// ============================================
// DB_RecipeProgram3 - Program 3
// Lines: 97
// CHUNKS: 5 x 100
// Generated by SpinningCam  [2026-09-29 00:05:30]
// !!! CONTINUOUS MOTION (CMD=2) - EXPERIMENTAL PLC ONLY !!!
// Load ONLY on the continuous-motion PLC build. A production PLC
// skips CMD=2 lines and jumps straight between the other points.
// T=0.045 s, corner tol=0.2 mm, F min=180, exact stop at >= 90 deg, stop slow-down=OFF
// CMD=2 lines: 76, exact corners: 0, slowed corners: 7 (+11 leaving), slowed stops: 0
// ============================================
//
// --- MAKINE AYARLARI ---
// Machine Origin  : X=0.0, Z=0.0
// Axis Direction  : X=NORMAL, Z=NORMAL
// Output Mode     : RADIUS
// G54 Offset      : X=0.0, Z=0.0
// Home            : X=-394.0, Z=-174.0
// Retract         : X=-10.0, Z=-10.0
//
// --- PARCA / BLANK ---
// Blank Radius    : 77.8 mm
// Blank Z Shift   : 0.0 mm
// Final Thickness : 0.8 mm
// Min Safety Gap  : 0.0 mm
//
// --- MANDREL POZISYON ---
// Mandrel Offset  : X=0.0, Z=0.0
// Mandrel Rot     : Rx=90.0, Ry=0.0, Rz=0.0
//
// --- OPERASYONLAR ---
// Op1: ROUGHING, 1 paso, T004, R=44.56mm, RPM=600.0, mm_min=900.0
// Op2: ROUGHING, 1 paso, T004, R=44.56mm, RPM=600.0, mm_min=900.0
// Op3: ROUGHING, 1 paso, T004, R=44.56mm, RPM=600.0, mm_min=900.0
// Op4: ROUGHING, 1 paso, T004, R=44.56mm, RPM=600.0, mm_min=900.0
// Op5: ROUGHING, 1 paso, T004, R=44.56mm, RPM=600.0, mm_min=900.0
// Op6: ROUGHING, 1 paso, T004, R=44.56mm, RPM=600.0, mm_min=800.0
// Op7: ROUGHING, 1 paso, T004, R=44.56mm, RPM=600.0, mm_min=800.0
// Op8: ROUGHING, 1 paso, T004, R=44.56mm, RPM=600.0, mm_min=800.0
// Op9: ROUGHING, 1 paso, T004, R=44.56mm, RPM=600.0, mm_min=800.0
// Op10: ROUGHING, 1 paso, T004, R=44.56mm, RPM=600.0, mm_min=800.0
// Op11: ROUGHING, 1 paso, T004, R=44.56mm, RPM=600.0, mm_min=800.0
// Op12: ROUGHING, 1 paso, T004, R=44.56mm, RPM=600.0, mm_min=800.0
// Op13: ROUGHING, 1 paso, T004, R=44.56mm, RPM=600.0, mm_min=1000.0
// Op14: ROUGHING, 1 paso, T004, R=44.56mm, RPM=600.0, mm_min=1000.0
// Op15: ROUGHING, 1 paso, T004, R=44.56mm, RPM=600.0, mm_min=1000.0
// Op16: ROUGHING, 1 paso, T004, R=44.56mm, RPM=600.0, mm_min=1000.0
// Op17: ROUGHING, 1 paso, T004, R=44.56mm, RPM=600.0, mm_min=1000.0
// Op18: ROUGHING, 1 paso, T004, R=44.56mm, RPM=600.0, mm_min=1000.0
// Op19: ROUGHING, 1 paso, T004, R=44.56mm, RPM=600.0, mm_min=1000.0
// Op20: ROUGHING, 1 paso, T004, R=44.56mm, RPM=600.0, mm_min=1000.0
// Op21: ROUGHING, 1 paso, T004, R=44.56mm, RPM=600.0, mm_min=1000.0
// Op22: ROUGHING, 1 paso, T004, R=44.56mm, RPM=600.0, mm_min=1000.0
// Op23: ROUGHING, 1 paso, T004, R=44.56mm, RPM=600.0, mm_min=1000.0
// Op24: ROUGHING, 1 paso, T004, R=44.56mm, RPM=600.0, mm_min=1000.0
// Op25: ROUGHING, 1 paso, T004, R=44.56mm, RPM=600.0, mm_min=1000.0
// Op26: ROUGHING, 1 paso, T004, R=44.56mm, RPM=600.0, mm_min=1000.0
// Op27: CUTTING, 1 paso, T006, R=20.0mm, RPM=500.0, mm_min=10.0
// Op28: ROUGHING, 1 paso, T004, R=44.56mm, RPM=600.0, mm_min=1000.0
// Op29: ROUGHING, 1 paso, T004, R=44.56mm, RPM=600.0, mm_min=1000.0
// Op30: ROUGHING, 1 paso, T004, R=44.56mm, RPM=600.0, mm_min=1000.0
// Op31: ROUGHING, 1 paso, T004, R=44.56mm, RPM=600.0, mm_min=1000.0
// Op32: ROUGHING, 1 paso, T004, R=44.56mm, RPM=600.0, mm_min=1000.0
// Op33: ROUGHING, 1 paso, T004, R=44.56mm, RPM=600.0, mm_min=1000.0
// Op34: ROUGHING, 1 paso, T004, R=44.56mm, RPM=600.0, mm_min=1000.0
// Op35: ROUGHING, 1 paso, T004, R=44.56mm, RPM=600.0, mm_min=1000.0
// Op36: ROUGHING, 1 paso, T004, R=44.56mm, RPM=600.0, mm_min=1500.0
// Op37: ROUGHING, 1 paso, T004, R=44.56mm, RPM=600.0, mm_min=1500.0
// Op38: ROUGHING, 1 paso, T004, R=44.56mm, RPM=600.0, mm_min=1500.0
// Op39: ROUGHING, 1 paso, T004, R=44.56mm, RPM=600.0, mm_min=1500.0
// Op40: ROUGHING, 1 paso, T004, R=44.56mm, RPM=600.0, mm_min=1500.0
// Op41: ROUGHING, 1 paso, T004, R=44.56mm, RPM=600.0, mm_min=1500.0
// Op42: ROUGHING, 1 paso, T004, R=44.56mm, RPM=600.0, mm_min=1500.0
// Op43: ROUGHING, 1 paso, T004, R=44.56mm, RPM=600.0, mm_min=1500.0
// Op44: ROUGHING, 1 paso, T004, R=44.56mm, RPM=600.0, mm_min=1500.0
// Op45: ROUGHING, 1 paso, T004, R=44.56mm, RPM=600.0, mm_min=1500.0
// Op46: ROUGHING, 1 paso, T004, R=44.56mm, RPM=600.0, mm_min=1500.0
// Op47: ROUGHING, 1 paso, T004, R=44.56mm, RPM=600.0, mm_min=1500.0
// Op48: ROUGHING, 1 paso, T004, R=44.56mm, RPM=600.0, mm_min=1500.0
// Op49: ROUGHING, 1 paso, T004, R=44.56mm, RPM=600.0, mm_min=1500.0
// Op50: ROUGHING, 1 paso, T004, R=44.56mm, RPM=600.0, mm_min=1500.0
// Op51: ROUGHING, 1 paso, T004, R=44.56mm, RPM=600.0, mm_min=1500.0
// Op52: ROUGHING, 1 paso, T004, R=44.56mm, RPM=600.0, mm_min=1500.0
// Op53: ROUGHING, 1 paso, T004, R=44.56mm, RPM=600.0, mm_min=1500.0
// Op54: ROUGHING, 1 paso, T004, R=44.56mm, RPM=600.0, mm_min=1500.0
// Op55: ROUGHING, 1 paso, T004, R=44.56mm, RPM=600.0, mm_min=1500.0
// Op56: ROUGHING, 1 paso, T004, R=44.56mm, RPM=600.0, mm_min=1500.0
// Op57: ROUGHING, 1 paso, T004, R=44.56mm, RPM=600.0, mm_min=1500.0
// Op58: ROUGHING, 1 paso, T004, R=44.56mm, RPM=600.0, mm_min=1500.0
// Op59: ROUGHING, 1 paso, T004, R=44.56mm, RPM=600.0, mm_min=1500.0
// Op60: ROUGHING, 1 paso, T004, R=44.56mm, RPM=800.0, mm_min=1500.0
// Op61: ROUGHING, 1 paso, T004, R=44.56mm, RPM=800.0, mm_min=800.0
// Op62: ROUGHING, 1 paso, T004, R=44.56mm, RPM=800.0, mm_min=800.0
// Op63: ROUGHING, 1 paso, T004, R=44.56mm, RPM=600.0, mm_min=1500.0
// Op64: ROUGHING, 1 paso, T004, R=44.56mm, RPM=600.0, mm_min=1500.0
// Op65: ROUGHING, 1 paso, T004, R=44.56mm, RPM=600.0, mm_min=1500.0
// Op66: ROUGHING, 1 paso, T004, R=44.56mm, RPM=600.0, mm_min=1500.0
// Op67: ROUGHING, 1 paso, T004, R=44.56mm, RPM=600.0, mm_min=1500.0
// Op68: ROUGHING, 1 paso, T004, R=44.56mm, RPM=600.0, mm_min=1500.0
// Op69: ROUGHING, 1 paso, T004, R=44.56mm, RPM=600.0, mm_min=1500.0
// Op70: ROUGHING, 1 paso, T004, R=44.56mm, RPM=600.0, mm_min=1500.0
// Op71: ROUGHING, 1 paso, T004, R=44.56mm, RPM=600.0, mm_min=1500.0
// Op72: ROUGHING, 1 paso, T004, R=44.56mm, RPM=600.0, mm_min=1000.0
// Op73: ROUGHING, 1 paso, T004, R=44.56mm, RPM=600.0, mm_min=1000.0
// Op74: ROUGHING, 1 paso, T004, R=44.56mm, RPM=600.0, mm_min=1000.0
// Op75: ROUGHING, 1 paso, T004, R=44.56mm, RPM=600.0, mm_min=1000.0
// Op76: ROUGHING, 1 paso, T004, R=44.56mm, RPM=600.0, mm_min=1500.0
// Op77: ROUGHING, 1 paso, T004, R=44.56mm, RPM=600.0, mm_min=1000.0
// Op78: ROUGHING, 1 paso, T004, R=44.56mm, RPM=600.0, mm_min=1000.0
// Op79: ROUGHING, 1 paso, T004, R=44.56mm, RPM=600.0, mm_min=1000.0
// Op80: ROUGHING, 1 paso, T004, R=44.56mm, RPM=600.0, mm_min=1000.0
// Op81: ROUGHING, 1 paso, T004, R=44.56mm, RPM=600.0, mm_min=1000.0
// Op82: ROUGHING, 1 paso, T004, R=44.56mm, RPM=600.0, mm_min=1000.0
// Op83: ROUGHING, 1 paso, T004, R=44.56mm, RPM=600.0, mm_min=1000.0
// Op84: ROUGHING, 1 paso, T004, R=44.56mm, RPM=600.0, mm_min=1000.0
// Op85: ROUGHING, 1 paso, T004, R=44.56mm, RPM=600.0, mm_min=1000.0
// Op86: ROUGHING, 1 paso, T004, R=44.56mm, RPM=600.0, mm_min=1000.0
// Op87: ROUGHING, 1 paso, T004, R=44.56mm, RPM=600.0, mm_min=1000.0
// Op88: ROUGHING, 1 paso, T004, R=44.56mm, RPM=600.0, mm_min=1000.0
// Op89: ROUGHING, 1 paso, T004, R=44.56mm, RPM=600.0, mm_min=1000.0
// Op90: ROUGHING, 1 paso, T004, R=44.56mm, RPM=600.0, mm_min=1000.0
// Op91: ROUGHING, 1 paso, T004, R=44.56mm, RPM=600.0, mm_min=1000.0
// Op92: ROUGHING, 1 paso, T004, R=44.56mm, RPM=600.0, mm_min=1000.0
// Op93: ROUGHING, 1 paso, T004, R=44.56mm, RPM=600.0, mm_min=1000.0
// Op94: ROUGHING, 1 paso, T004, R=44.56mm, RPM=600.0, mm_min=1000.0
// Op95: ROUGHING, 1 paso, T004, R=44.56mm, RPM=600.0, mm_min=1000.0
// Op96: ROUGHING, 1 paso, T004, R=44.56mm, RPM=600.0, mm_min=1000.0
// Op97: ROUGHING, 1 paso, T004, R=44.56mm, RPM=600.0, mm_min=1000.0
// Op98: ROUGHING, 1 paso, T004, R=44.56mm, RPM=600.0, mm_min=1000.0
// Op99: ROUGHING, 1 paso, T004, R=44.56mm, RPM=600.0, mm_min=1000.0
// Op100: ROUGHING, 1 paso, T004, R=44.56mm, RPM=600.0, mm_min=1000.0
// Op101: ROUGHING, 1 paso, T004, R=44.56mm, RPM=600.0, mm_min=1000.0
// Op102: ROUGHING, 1 paso, T004, R=44.56mm, RPM=600.0, mm_min=1000.0
// Op103: ROUGHING, 1 paso, T004, R=44.56mm, RPM=600.0, mm_min=1000.0
// Op104: ROUGHING, 1 paso, T004, R=44.56mm, RPM=600.0, mm_min=1000.0
// Op105: ROUGHING, 1 paso, T004, R=44.56mm, RPM=600.0, mm_min=1000.0
// Op106: ROUGHING, 1 paso, T004, R=44.56mm, RPM=600.0, mm_min=1000.0
// Op107: ROUGHING, 1 paso, T004, R=44.56mm, RPM=600.0, mm_min=1000.0
// Op108: ROUGHING, 1 paso, T004, R=44.56mm, RPM=600.0, mm_min=1000.0
// Op109: ROUGHING, 1 paso, T004, R=44.56mm, RPM=600.0, mm_min=1000.0
// Op110: ROUGHING, 1 paso, T004, R=44.56mm, RPM=600.0, mm_min=1000.0
// Op111: ROUGHING, 1 paso, T004, R=44.56mm, RPM=600.0, mm_min=1000.0
// Op112: ROUGHING, 1 paso, T004, R=44.56mm, RPM=600.0, mm_min=1000.0
// Op113: ROUGHING, 1 paso, T004, R=44.56mm, RPM=600.0, mm_min=1000.0
// Op114: ROUGHING, 1 paso, T004, R=44.56mm, RPM=600.0, mm_min=1000.0
// Op115: ROUGHING, 1 paso, T004, R=44.56mm, RPM=600.0, mm_min=1000.0
// Op116: ROUGHING, 1 paso, T004, R=44.56mm, RPM=600.0, mm_min=1000.0
// Op117: ROUGHING, 1 paso, T004, R=44.56mm, RPM=600.0, mm_min=1000.0
// Op118: ROUGHING, 1 paso, T004, R=44.56mm, RPM=600.0, mm_min=1000.0
// Op119: ROUGHING, 1 paso, T004, R=44.56mm, RPM=600.0, mm_min=1000.0
// Op120: ROUGHING, 1 paso, T004, R=44.56mm, RPM=600.0, mm_min=1000.0
// Op121: ROUGHING, 1 paso, T004, R=44.56mm, RPM=600.0, mm_min=1000.0
// Op122: ROUGHING, 1 paso, T004, R=44.56mm, RPM=600.0, mm_min=1000.0
// Op123: ROUGHING, 1 paso, T004, R=44.56mm, RPM=600.0, mm_min=1000.0
// Op124: ROUGHING, 1 paso, T004, R=44.56mm, RPM=600.0, mm_min=1000.0
// Op125: ROUGHING, 1 paso, T004, R=44.56mm, RPM=600.0, mm_min=1000.0
// Op126: ROUGHING, 1 paso, T004, R=44.56mm, RPM=600.0, mm_min=1000.0
// Op127: ROUGHING, 1 paso, T004, R=44.56mm, RPM=600.0, mm_min=1000.0
// Op128: ROUGHING, 1 paso, T004, R=44.56mm, RPM=600.0, mm_min=1000.0
// Op129: CUTTING, 1 paso, T006, R=20.0mm, RPM=500.0, mm_min=7.0
// Op130: ROUGHING, 1 paso, T004, R=44.56mm, RPM=600.0, mm_min=1000.0
// Op131: ROUGHING, 1 paso, T004, R=44.56mm, RPM=600.0, mm_min=1000.0
// Op132: ROUGHING, 1 paso, T004, R=44.56mm, RPM=600.0, mm_min=1000.0
// Op133: ROUGHING, 1 paso, T004, R=44.56mm, RPM=600.0, mm_min=1000.0
// Op134: ROUGHING, 1 paso, T004, R=44.56mm, RPM=600.0, mm_min=1000.0
// Op135: ROUGHING, 1 paso, T004, R=44.56mm, RPM=600.0, mm_min=1000.0
// Op136: ROUGHING, 1 paso, T004, R=44.56mm, RPM=600.0, mm_min=1000.0
// Op137: ROUGHING, 1 paso, T004, R=44.56mm, RPM=600.0, mm_min=400.0
// Op138: ROUGHING, 1 paso, T004, R=44.56mm, RPM=600.0, mm_min=400.0
// Op139: ROUGHING, 1 paso, T004, R=44.56mm, RPM=600.0, mm_min=400.0
// Op140: ROUGHING, 1 paso, T004, R=44.56mm, RPM=600.0, mm_min=1000.0
// Op141: ROUGHING, 1 paso, T004, R=44.56mm, RPM=600.0, mm_min=400.0
// Op142: ROUGHING, 1 paso, T004, R=44.56mm, RPM=600.0, mm_min=400.0
// Op143: ROUGHING, 1 paso, T004, R=44.56mm, RPM=600.0, mm_min=400.0
// Op144: ROUGHING, 1 paso, T004, R=44.56mm, RPM=600.0, mm_min=400.0
// Op145: ROUGHING, 1 paso, T004, R=44.56mm, RPM=600.0, mm_min=400.0
// Op146: ROUGHING, 1 paso, T004, R=44.56mm, RPM=600.0, mm_min=400.0
// Op147: ROUGHING, 1 paso, T004, R=44.56mm, RPM=600.0, mm_min=400.0
// Op148: ROUGHING, 1 paso, T004, R=44.56mm, RPM=600.0, mm_min=400.0
// Op149: ROUGHING, 1 paso, T004, R=44.56mm, RPM=600.0, mm_min=400.0
// Op150: ROUGHING, 1 paso, T004, R=44.56mm, RPM=600.0, mm_min=400.0
// Op151: ROUGHING, 1 paso, T004, R=44.56mm, RPM=600.0, mm_min=400.0
// Op152: ROUGHING, 1 paso, T004, R=44.56mm, RPM=600.0, mm_min=400.0
// Op153: ROUGHING, 1 paso, T004, R=44.56mm, RPM=600.0, mm_min=400.0
// Op154: ROUGHING, 1 paso, T004, R=44.56mm, RPM=600.0, mm_min=400.0
// Op155: ROUGHING, 1 paso, T004, R=44.56mm, RPM=600.0, mm_min=400.0
// Op156: ROUGHING, 1 paso, T004, R=44.56mm, RPM=600.0, mm_min=400.0
// Op157: ROUGHING, 1 paso, T004, R=44.56mm, RPM=600.0, mm_min=400.0
// Op158: ROUGHING, 1 paso, T004, R=44.56mm, RPM=600.0, mm_min=400.0
// Op159: ROUGHING, 1 paso, T004, R=44.56mm, RPM=600.0, mm_min=400.0
// Op160: ROUGHING, 1 paso, T004, R=44.56mm, RPM=600.0, mm_min=400.0
// Op161: ROUGHING, 1 paso, T004, R=44.56mm, RPM=600.0, mm_min=400.0
// Op162: ROUGHING, 1 paso, T004, R=44.56mm, RPM=600.0, mm_min=400.0
// Op163: ROUGHING, 1 paso, T004, R=44.56mm, RPM=600.0, mm_min=400.0
// Op164: ROUGHING, 1 paso, T004, R=44.56mm, RPM=600.0, mm_min=400.0
// Op165: ROUGHING, 1 paso, T004, R=44.56mm, RPM=600.0, mm_min=400.0
// Op166: ROUGHING, 1 paso, T004, R=44.56mm, RPM=600.0, mm_min=400.0
// Op167: ROUGHING, 1 paso, T004, R=44.56mm, RPM=800.0, mm_min=400.0
// Op168: ROUGHING, 1 paso, T004, R=44.56mm, RPM=800.0, mm_min=400.0
// Op169: ROUGHING, 1 paso, T004, R=44.56mm, RPM=800.0, mm_min=400.0
// Op170: ROUGHING, 1 paso, T004, R=44.56mm, RPM=800.0, mm_min=400.0
// Op171: ROUGHING, 1 paso, T004, R=44.56mm, RPM=800.0, mm_min=400.0
// Op172: ROUGHING, 1 paso, T004, R=44.56mm, RPM=800.0, mm_min=400.0
// Op173: ROUGHING, 1 paso, T004, R=44.56mm, RPM=800.0, mm_min=400.0
// Op174: ROUGHING, 1 paso, T004, R=44.56mm, RPM=800.0, mm_min=400.0
// Op175: ROUGHING, 1 paso, T004, R=44.56mm, RPM=800.0, mm_min=400.0
// Op176: ROUGHING, 1 paso, T004, R=44.56mm, RPM=800.0, mm_min=400.0
// Op177: ROUGHING, 1 paso, T004, R=44.56mm, RPM=800.0, mm_min=400.0
// Op178: ROUGHING, 1 paso, T004, R=44.56mm, RPM=800.0, mm_min=400.0
// Op179: ROUGHING, 1 paso, T004, R=44.56mm, RPM=800.0, mm_min=400.0
// Op180: ROUGHING, 1 paso, T004, R=44.56mm, RPM=800.0, mm_min=400.0
// Op181: ROUGHING, 1 paso, T004, R=44.56mm, RPM=800.0, mm_min=400.0
// Op182: ROUGHING, 1 paso, T004, R=44.56mm, RPM=800.0, mm_min=400.0
// Op183: ROUGHING, 1 paso, T004, R=44.56mm, RPM=800.0, mm_min=400.0
// ============================================

DATA_BLOCK "DB_RecipeProgram3"
{ S7_Optimized_Access := 'FALSE' }
VERSION : 0.2
UNLINKED
NON_RETAIN
    VAR
        Header : "RecipeHeader";
        Lines1 : Array[0..99] of "RecipeLine";  // global lines 0..99
        Lines2 : Array[0..99] of "RecipeLine";  // global lines 100..199
        Lines3 : Array[0..99] of "RecipeLine";  // global lines 200..299
        Lines4 : Array[0..99] of "RecipeLine";  // global lines 300..399
        Lines5 : Array[0..99] of "RecipeLine";  // global lines 400..499
    END_VAR
BEGIN
    // Header
    Header.sName := 'Program 3';
    Header.LineCount := 97;
    Header.Valid := TRUE;
    Header.PreScanned := FALSE;
    Header.MinX := 173.498;
    Header.MaxX := 273.206;
    Header.MinZ := 74.000;
    Header.MaxZ := 252.648;

    // --- Tool table (CAM-authored) ---
    Header.ProvidesToolConfig := TRUE;
    Header.ToolCount := 4;
    Header.AutoCalcAngles := FALSE;
    Header.ToolCode_List[1] := 4;
    Header.ToolCode_List[2] := 5;
    Header.ToolCode_List[3] := 6;
    Header.ToolCode_List[4] := 7;
    Header.ToolAngle_List[1] := 0.0;
    Header.ToolAngle_List[2] := 120.0;
    Header.ToolAngle_List[3] := 240.0;
    Header.ToolAngle_List[4] := 360.0;

    // --- Integrity ---
    // Order-sensitive sum over CMD+Param+F of lines 0..LineCount-1.
    // The PLC recomputes it after reassembling the chunks and refuses
    // to run on a mismatch (16#0316). X/Z are excluded on purpose:
    // float32-vs-float64 rounding would eventually cry wolf.
    Header.ProvidesChecksum := TRUE;
    Header.Checksum := 2953499;

    // Recipe Lines (97 total)

    // --- Lines1 (global lines 0..96) ---
    Lines1[0].X := 0.000; Lines1[0].Z := 0.000; Lines1[0].F := 0; Lines1[0].CMD := 40; Lines1[0].Param := 80; // Cylinder GOTO P80
    Lines1[1].X := 0.000; Lines1[1].Z := 0.000; Lines1[1].F := 0; Lines1[1].CMD := 10; Lines1[1].Param := 4; // Tool Change T4
    Lines1[2].X := 0.000; Lines1[2].Z := 0.000; Lines1[2].F := 0; Lines1[2].CMD := 20; Lines1[2].Param := 60; // Spindle ON 600 RPM
    Lines1[3].X := 0.000; Lines1[3].Z := 0.000; Lines1[3].F := 0; Lines1[3].CMD := 41; Lines1[3].Param := 1; // M41 (Clamp On) P1 [Op1 P1]
    Lines1[4].X := 272.912; Lines1[4].Z := 176.000; Lines1[4].F := 0; Lines1[4].CMD := 0; Lines1[4].Param := 0; // G0 Rapid [Op1 P1]
    Lines1[5].X := 272.901; Lines1[5].Z := 181.258; Lines1[5].F := 900; Lines1[5].CMD := 2; Lines1[5].Param := 0; // G1 Continuous [Op1 P1]
    Lines1[6].X := 272.695; Lines1[6].Z := 182.343; Lines1[6].F := 737; Lines1[6].CMD := 2; Lines1[6].Param := 0; // G1 Continuous [Op1 P1]
    Lines1[7].X := 272.111; Lines1[7].Z := 183.280; Lines1[7].F := 737; Lines1[7].CMD := 2; Lines1[7].Param := 0; // G1 Continuous [Op1 P1]
    Lines1[8].X := 271.227; Lines1[8].Z := 183.943; Lines1[8].F := 735; Lines1[8].CMD := 2; Lines1[8].Param := 0; // G1 Continuous [Op1 P1]
    Lines1[9].X := 270.164; Lines1[9].Z := 184.240; Lines1[9].F := 735; Lines1[9].CMD := 2; Lines1[9].Param := 0; // G1 Continuous [Op1 P1]
    Lines1[10].X := 178.498; Lines1[10].Z := 192.302; Lines1[10].F := 900; Lines1[10].CMD := 2; Lines1[10].Param := 0; // G1 Continuous [Op1 P1]
    Lines1[11].X := 173.498; Lines1[11].Z := 187.302; Lines1[11].F := 0; Lines1[11].CMD := 0; Lines1[11].Param := 0; // G0 Rapid [Op1 P1]
    Lines1[12].X := 173.498; Lines1[12].Z := 187.302; Lines1[12].F := 0; Lines1[12].CMD := 41; Lines1[12].Param := 2; // M41 (Clamp On) P2 [Op2 P1]
    Lines1[13].X := 273.001; Lines1[13].Z := 182.538; Lines1[13].F := 0; Lines1[13].CMD := 0; Lines1[13].Param := 0; // G0 Rapid [Op2 P1]
    Lines1[14].X := 272.998; Lines1[14].Z := 183.142; Lines1[14].F := 900; Lines1[14].CMD := 2; Lines1[14].Param := 0; // G1 Continuous [Op2 P1]
    Lines1[15].X := 272.803; Lines1[15].Z := 184.197; Lines1[15].F := 859; Lines1[15].CMD := 2; Lines1[15].Param := 0; // G1 Continuous [Op2 P1]
    Lines1[16].X := 272.418; Lines1[16].Z := 184.905; Lines1[16].F := 859; Lines1[16].CMD := 2; Lines1[16].Param := 0; // G1 Continuous [Op2 P1]
    Lines1[17].X := 271.639; Lines1[17].Z := 185.643; Lines1[17].F := 756; Lines1[17].CMD := 2; Lines1[17].Param := 0; // G1 Continuous [Op2 P1]
    Lines1[18].X := 270.650; Lines1[18].Z := 186.059; Lines1[18].F := 756; Lines1[18].CMD := 2; Lines1[18].Param := 0; // G1 Continuous [Op2 P1]
    Lines1[19].X := 180.388; Lines1[19].Z := 206.156; Lines1[19].F := 900; Lines1[19].CMD := 2; Lines1[19].Param := 0; // G1 Continuous [Op2 P1]
    Lines1[20].X := 272.995; Lines1[20].Z := 184.077; Lines1[20].F := 0; Lines1[20].CMD := 0; Lines1[20].Param := 0; // G0 Rapid [Op3 P1]
    Lines1[21].X := 272.992; Lines1[21].Z := 184.868; Lines1[21].F := 900; Lines1[21].CMD := 2; Lines1[21].Param := 0; // G1 Continuous [Op3 P1]
    Lines1[22].X := 272.879; Lines1[22].Z := 185.674; Lines1[22].F := 854; Lines1[22].CMD := 2; Lines1[22].Param := 0; // G1 Continuous [Op3 P1]
    Lines1[23].X := 272.402; Lines1[23].Z := 186.645; Lines1[23].F := 750; Lines1[23].CMD := 2; Lines1[23].Param := 0; // G1 Continuous [Op3 P1]
    Lines1[24].X := 271.611; Lines1[24].Z := 187.383; Lines1[24].F := 750; Lines1[24].CMD := 2; Lines1[24].Param := 0; // G1 Continuous [Op3 P1]
    Lines1[25].X := 270.873; Lines1[25].Z := 187.725; Lines1[25].F := 856; Lines1[25].CMD := 2; Lines1[25].Param := 0; // G1 Continuous [Op3 P1]
    Lines1[26].X := 182.286; Lines1[26].Z := 214.928; Lines1[26].F := 900; Lines1[26].CMD := 2; Lines1[26].Param := 0; // G1 Continuous [Op3 P1]
    Lines1[27].X := 273.006; Lines1[27].Z := 181.000; Lines1[27].F := 0; Lines1[27].CMD := 0; Lines1[27].Param := 0; // G0 Rapid [Op4 P1]
    Lines1[28].X := 272.984; Lines1[28].Z := 186.988; Lines1[28].F := 900; Lines1[28].CMD := 2; Lines1[28].Param := 0; // G1 Continuous [Op4 P1]
    Lines1[29].X := 272.871; Lines1[29].Z := 187.795; Lines1[29].F := 900; Lines1[29].CMD := 2; Lines1[29].Param := 0; // G1 Continuous [Op4 P1]
    Lines1[30].X := 272.544; Lines1[30].Z := 188.542; Lines1[30].F := 852; Lines1[30].CMD := 2; Lines1[30].Param := 0; // G1 Continuous [Op4 P1]
    Lines1[31].X := 271.820; Lines1[31].Z := 189.350; Lines1[31].F := 852; Lines1[31].CMD := 2; Lines1[31].Param := 0; // G1 Continuous [Op4 P1]
    Lines1[32].X := 271.113; Lines1[32].Z := 189.757; Lines1[32].F := 853; Lines1[32].CMD := 2; Lines1[32].Param := 0; // G1 Continuous [Op4 P1]
    Lines1[33].X := 185.053; Lines1[33].Z := 224.685; Lines1[33].F := 900; Lines1[33].CMD := 2; Lines1[33].Param := 0; // G1 Continuous [Op4 P1]
    Lines1[34].X := 273.006; Lines1[34].Z := 181.000; Lines1[34].F := 0; Lines1[34].CMD := 0; Lines1[34].Param := 0; // G0 Rapid [Op5 P1]
    Lines1[35].X := 272.980; Lines1[35].Z := 188.100; Lines1[35].F := 900; Lines1[35].CMD := 2; Lines1[35].Param := 0; // G1 Continuous [Op5 P1]
    Lines1[36].X := 272.859; Lines1[36].Z := 188.935; Lines1[36].F := 900; Lines1[36].CMD := 2; Lines1[36].Param := 0; // G1 Continuous [Op5 P1]
    Lines1[37].X := 272.509; Lines1[37].Z := 189.704; Lines1[37].F := 900; Lines1[37].CMD := 2; Lines1[37].Param := 0; // G1 Continuous [Op5 P1]
    Lines1[38].X := 271.959; Lines1[38].Z := 190.344; Lines1[38].F := 900; Lines1[38].CMD := 2; Lines1[38].Param := 0; // G1 Continuous [Op5 P1]
    Lines1[39].X := 271.253; Lines1[39].Z := 190.806; Lines1[39].F := 900; Lines1[39].CMD := 2; Lines1[39].Param := 0; // G1 Continuous [Op5 P1]
    Lines1[40].X := 187.038; Lines1[40].Z := 230.259; Lines1[40].F := 900; Lines1[40].CMD := 2; Lines1[40].Param := 0; // G1 Continuous [Op5 P1]
    Lines1[41].X := 273.106; Lines1[41].Z := 181.000; Lines1[41].F := 0; Lines1[41].CMD := 0; Lines1[41].Param := 0; // G0 Rapid [Op6 P1]
    Lines1[42].X := 273.076; Lines1[42].Z := 189.172; Lines1[42].F := 800; Lines1[42].CMD := 2; Lines1[42].Param := 0; // G1 Continuous [Op6 P1]
    Lines1[43].X := 272.962; Lines1[43].Z := 189.982; Lines1[43].F := 800; Lines1[43].CMD := 2; Lines1[43].Param := 0; // G1 Continuous [Op6 P1]
    Lines1[44].X := 272.633; Lines1[44].Z := 190.731; Lines1[44].F := 800; Lines1[44].CMD := 2; Lines1[44].Param := 0; // G1 Continuous [Op6 P1]
    Lines1[45].X := 272.113; Lines1[45].Z := 191.364; Lines1[45].F := 800; Lines1[45].CMD := 2; Lines1[45].Param := 0; // G1 Continuous [Op6 P1]
    Lines1[46].X := 271.442; Lines1[46].Z := 191.832; Lines1[46].F := 800; Lines1[46].CMD := 2; Lines1[46].Param := 0; // G1 Continuous [Op6 P1]
    Lines1[47].X := 188.492; Lines1[47].Z := 234.247; Lines1[47].F := 800; Lines1[47].CMD := 2; Lines1[47].Param := 0; // G1 Continuous [Op6 P1]
    Lines1[48].X := 273.106; Lines1[48].Z := 181.000; Lines1[48].F := 0; Lines1[48].CMD := 0; Lines1[48].Param := 0; // G0 Rapid [Op7 P1]
    Lines1[49].X := 273.072; Lines1[49].Z := 190.278; Lines1[49].F := 800; Lines1[49].CMD := 2; Lines1[49].Param := 0; // G1 Continuous [Op7 P1]
    Lines1[50].X := 272.949; Lines1[50].Z := 191.119; Lines1[50].F := 800; Lines1[50].CMD := 2; Lines1[50].Param := 0; // G1 Continuous [Op7 P1]
    Lines1[51].X := 272.737; Lines1[51].Z := 191.646; Lines1[51].F := 800; Lines1[51].CMD := 2; Lines1[51].Param := 0; // G1 Continuous [Op7 P1]
    Lines1[52].X := 272.244; Lines1[52].Z := 192.337; Lines1[52].F := 800; Lines1[52].CMD := 2; Lines1[52].Param := 0; // G1 Continuous [Op7 P1]
    Lines1[53].X := 271.576; Lines1[53].Z := 192.863; Lines1[53].F := 800; Lines1[53].CMD := 2; Lines1[53].Param := 0; // G1 Continuous [Op7 P1]
    Lines1[54].X := 190.869; Lines1[54].Z := 239.630; Lines1[54].F := 800; Lines1[54].CMD := 2; Lines1[54].Param := 0; // G1 Continuous [Op7 P1]
    Lines1[55].X := 273.106; Lines1[55].Z := 181.000; Lines1[55].F := 0; Lines1[55].CMD := 0; Lines1[55].Param := 0; // G0 Rapid [Op8 P1]
    Lines1[56].X := 273.068; Lines1[56].Z := 191.382; Lines1[56].F := 800; Lines1[56].CMD := 2; Lines1[56].Param := 0; // G1 Continuous [Op8 P1]
    Lines1[57].X := 273.008; Lines1[57].Z := 191.971; Lines1[57].F := 800; Lines1[57].CMD := 2; Lines1[57].Param := 0; // G1 Continuous [Op8 P1]
    Lines1[58].X := 272.703; Lines1[58].Z := 192.805; Lines1[58].F := 800; Lines1[58].CMD := 2; Lines1[58].Param := 0; // G1 Continuous [Op8 P1]
    Lines1[59].X := 272.169; Lines1[59].Z := 193.513; Lines1[59].F := 800; Lines1[59].CMD := 2; Lines1[59].Param := 0; // G1 Continuous [Op8 P1]
    Lines1[60].X := 271.707; Lines1[60].Z := 193.884; Lines1[60].F := 800; Lines1[60].CMD := 2; Lines1[60].Param := 0; // G1 Continuous [Op8 P1]
    Lines1[61].X := 193.471; Lines1[61].Z := 244.882; Lines1[61].F := 800; Lines1[61].CMD := 2; Lines1[61].Param := 0; // G1 Continuous [Op8 P1]
    Lines1[62].X := 273.206; Lines1[62].Z := 181.000; Lines1[62].F := 0; Lines1[62].CMD := 0; Lines1[62].Param := 0; // G0 Rapid [Op9 P1]
    Lines1[63].X := 273.164; Lines1[63].Z := 192.448; Lines1[63].F := 800; Lines1[63].CMD := 2; Lines1[63].Param := 0; // G1 Continuous [Op9 P1]
    Lines1[64].X := 273.108; Lines1[64].Z := 193.017; Lines1[64].F := 800; Lines1[64].CMD := 2; Lines1[64].Param := 0; // G1 Continuous [Op9 P1]
    Lines1[65].X := 272.824; Lines1[65].Z := 193.825; Lines1[65].F := 800; Lines1[65].CMD := 2; Lines1[65].Param := 0; // G1 Continuous [Op9 P1]
    Lines1[66].X := 272.323; Lines1[66].Z := 194.520; Lines1[66].F := 800; Lines1[66].CMD := 2; Lines1[66].Param := 0; // G1 Continuous [Op9 P1]
    Lines1[67].X := 271.888; Lines1[67].Z := 194.892; Lines1[67].F := 800; Lines1[67].CMD := 2; Lines1[67].Param := 0; // G1 Continuous [Op9 P1]
    Lines1[68].X := 263.922; Lines1[68].Z := 201.440; Lines1[68].F := 800; Lines1[68].CMD := 2; Lines1[68].Param := 0; // G1 Continuous [Op9 P1]
    Lines1[69].X := 256.044; Lines1[69].Z := 207.677; Lines1[69].F := 800; Lines1[69].CMD := 2; Lines1[69].Param := 0; // G1 Continuous [Op9 P1]
    Lines1[70].X := 247.858; Lines1[70].Z := 213.913; Lines1[70].F := 800; Lines1[70].CMD := 2; Lines1[70].Param := 0; // G1 Continuous [Op9 P1]
    Lines1[71].X := 238.542; Lines1[71].Z := 220.721; Lines1[71].F := 800; Lines1[71].CMD := 2; Lines1[71].Param := 0; // G1 Continuous [Op9 P1]
    Lines1[72].X := 230.121; Lines1[72].Z := 226.621; Lines1[72].F := 800; Lines1[72].CMD := 2; Lines1[72].Param := 0; // G1 Continuous [Op9 P1]
    Lines1[73].X := 221.589; Lines1[73].Z := 232.363; Lines1[73].F := 800; Lines1[73].CMD := 2; Lines1[73].Param := 0; // G1 Continuous [Op9 P1]
    Lines1[74].X := 212.946; Lines1[74].Z := 237.946; Lines1[74].F := 800; Lines1[74].CMD := 2; Lines1[74].Param := 0; // G1 Continuous [Op9 P1]
    Lines1[75].X := 204.192; Lines1[75].Z := 243.372; Lines1[75].F := 800; Lines1[75].CMD := 2; Lines1[75].Param := 0; // G1 Continuous [Op9 P1]
    Lines1[76].X := 195.326; Lines1[76].Z := 248.639; Lines1[76].F := 800; Lines1[76].CMD := 2; Lines1[76].Param := 0; // G1 Continuous [Op9 P1]
    Lines1[77].X := 273.206; Lines1[77].Z := 181.000; Lines1[77].F := 0; Lines1[77].CMD := 0; Lines1[77].Param := 0; // G0 Rapid [Op10 P1]
    Lines1[78].X := 273.164; Lines1[78].Z := 192.546; Lines1[78].F := 800; Lines1[78].CMD := 2; Lines1[78].Param := 0; // G1 Continuous [Op10 P1]
    Lines1[79].X := 273.102; Lines1[79].Z := 193.143; Lines1[79].F := 800; Lines1[79].CMD := 2; Lines1[79].Param := 0; // G1 Continuous [Op10 P1]
    Lines1[80].X := 272.922; Lines1[80].Z := 193.717; Lines1[80].F := 800; Lines1[80].CMD := 2; Lines1[80].Param := 0; // G1 Continuous [Op10 P1]
    Lines1[81].X := 272.448; Lines1[81].Z := 194.481; Lines1[81].F := 800; Lines1[81].CMD := 2; Lines1[81].Param := 0; // G1 Continuous [Op10 P1]
    Lines1[82].X := 272.014; Lines1[82].Z := 194.897; Lines1[82].F := 800; Lines1[82].CMD := 2; Lines1[82].Param := 0; // G1 Continuous [Op10 P1]
    Lines1[83].X := 264.393; Lines1[83].Z := 201.861; Lines1[83].F := 800; Lines1[83].CMD := 2; Lines1[83].Param := 0; // G1 Continuous [Op10 P1]
    Lines1[84].X := 256.844; Lines1[84].Z := 208.508; Lines1[84].F := 800; Lines1[84].CMD := 2; Lines1[84].Param := 0; // G1 Continuous [Op10 P1]
    Lines1[85].X := 248.987; Lines1[85].Z := 215.172; Lines1[85].F := 800; Lines1[85].CMD := 2; Lines1[85].Param := 0; // G1 Continuous [Op10 P1]
    Lines1[86].X := 241.012; Lines1[86].Z := 221.683; Lines1[86].F := 800; Lines1[86].CMD := 2; Lines1[86].Param := 0; // G1 Continuous [Op10 P1]
    Lines1[87].X := 231.723; Lines1[87].Z := 228.960; Lines1[87].F := 800; Lines1[87].CMD := 2; Lines1[87].Param := 0; // G1 Continuous [Op10 P1]
    Lines1[88].X := 223.491; Lines1[88].Z := 235.145; Lines1[88].F := 800; Lines1[88].CMD := 2; Lines1[88].Param := 0; // G1 Continuous [Op10 P1]
    Lines1[89].X := 215.141; Lines1[89].Z := 241.177; Lines1[89].F := 800; Lines1[89].CMD := 2; Lines1[89].Param := 0; // G1 Continuous [Op10 P1]
    Lines1[90].X := 206.671; Lines1[90].Z := 247.058; Lines1[90].F := 800; Lines1[90].CMD := 2; Lines1[90].Param := 0; // G1 Continuous [Op10 P1]
    Lines1[91].X := 198.293; Lines1[91].Z := 252.648; Lines1[91].F := 800; Lines1[91].CMD := 2; Lines1[91].Param := 0; // G1 Continuous [Op10 P1]
    Lines1[92].X := 198.293; Lines1[92].Z := 74.000; Lines1[92].F := 0; Lines1[92].CMD := 0; Lines1[92].Param := 0; // G0 Rapid [Op10 P1]
    Lines1[93].X := 174.000; Lines1[93].Z := 74.000; Lines1[93].F := 0; Lines1[93].CMD := 0; Lines1[93].Param := 0; // G0 Rapid [Op10 P1]
    Lines1[94].X := 174.000; Lines1[94].Z := 74.000; Lines1[94].F := 0; Lines1[94].CMD := 21; Lines1[94].Param := 0; // Spindle OFF [Op10 P1]
    Lines1[95].X := 174.000; Lines1[95].Z := 74.000; Lines1[95].F := 0; Lines1[95].CMD := 21; Lines1[95].Param := 0; // Spindle OFF
    Lines1[96].X := 0.000; Lines1[96].Z := 0.000; Lines1[96].F := 0; Lines1[96].CMD := 99; Lines1[96].Param := 0; // Program END
END_DATA_BLOCK